(* PLC project tank, Dassault Systèmes ControlBuild 2024x *)
(* stored: creationDateTime 2023-10-03T11:13:04-01:00 *)

(* This module simulates the behaviour of the level in a tank. The input data for draining and filling are analog flows. *)
FUNCTION_BLOCK equipment_library.tank
  VAR_INPUT
    inletFlow : REAL := 0.0;
    outletFlow : REAL := 0.0;
  END_VAR
  VAR_OUTPUT
    tankLevel : REAL := 0.0;
  END_VAR
  VAR
    percent : REAL := 0.0;
  END_VAR
  VAR CONSTANT
    capacity : REAL := 1000.0;
  END_VAR
  VAR
    d_level : BOOL := false;
    v_d_level : REAL := 0.0;
  END_VAR


ACTION C_source_code:
/* -----------------------------------------------------------------	*/
/* Type : Model of Operative Behaviour					*/
/* Catégorie :   batch							*/
/* Author : Dassault Systemes						*/
/* Update date : June 2010							*/
/* -----------------------------------------------------------------	*/
/* This module simulates the behaviour of the level in a tank.	*/
/* The input data for draining and filling are analog flows.		*/
/* ----------------------------------------------------------------	*/

if (d_level ) tankLevel = v_d_level;	/* fault */
else  {
	/* compute level */
	tankLevel = tankLevel + inletFlow - outletFlow;

	/* bound level */
	if ( tankLevel >= capacity ) tankLevel = capacity;
	if ( tankLevel <= 0.0 ) tankLevel = 0.0; 	
}

/* ----------------------------------------------------------------	*/
/* Compute the percentage of filling					*/
/* ----------------------------------------------------------------	*/
if (capacity != 0.0) percent = ((tankLevel / capacity)*100);
END_ACTION
END_FUNCTION_BLOCK
